(* IEC 61131-3 sources: crb-codesys/generation/scripts/repoeval/轴控/FB105_轴控制集/FB50_虚轴控制/FB104_全局变量2, 13 files *)

(* ---- G01_调模A轴.st ---- *)
VAR_GLOBAL
	FB_AxisControl_调模A轴: FB_轴控块;

//轴触发类
	b调模A轴正向点动: BOOL;
	b调模A轴反向点动: BOOL;
	b调模A轴正向寸动: BOOL;
	b调模A轴反向寸动: BOOL;
	b调模A轴停止触发: BOOL;
	b调模A轴复位触发: BOOL;
	b调模A轴绝对运动触发: BOOL;
	b调模A轴相对运动触发: BOOL;
	b调模A轴速度模式触发: BOOL;
	b调模A轴启用限位: BOOL;

//轴状态类
    b调模A轴通讯OK: BOOL;
	b调模A轴使能OK: BOOL;
	b调模A轴停止完成: BOOL;
	b调模A轴绝对运动完成: BOOL;
	b调模A轴相对运动完成: BOOL;
	b调模A轴速度模式Busy: BOOL;
	b调模A轴寸动模式Busy: BOOL;
	b调模A轴点动模式Busy: BOOL;
	b调模A轴绝对模式Busy: BOOL;
	b调模A轴相对模式Busy: BOOL;
	b调模A轴错误: BOOL;
	b调模A轴加速中: BOOL;
	b调模A轴减速中: BOOL;
    b调模A轴停止中: BOOL;

//数据给定类
	r调模A轴点动速度给定: LREAL;
	r调模A轴绝对运动速度给定: LREAL;
	r调模A轴相对运动速度给定: LREAL;
	r调模A轴速度模式速度给定: LREAL;
	r调模A轴寸动速度给定: LREAL;

	r调模A轴绝对运动位置给定: LREAL;
	r调模A轴相对运动位置给定: LREAL;
	r调模A轴寸动位置给定: LREAL;

//数据读取类
    r调模A轴当前位置: LREAL;
	r调模A轴当前速度: LREAL;
	r调模A轴当前扭矩: LREAL;

//其它类
    b调模A轴回零触发: BOOL;
    b调模A轴回零Busy: BOOL;
    b调模A轴回零完成: BOOL;
END_VAR

//HMI_PLC_BOOL映射
VAR_GLOBAL
	HMI_b调模A轴断使能 	 AT %MX300.0: BOOL;
	HMI_b调模A轴单独回原 AT %MX300.1: BOOL;
	HMI_b调模A轴正向点动 AT %MX300.2: BOOL;
    HMI_b调模A轴反向点动 AT %MX300.3: BOOL;

	HMI_b调模A轴去工作位 AT %MX300.4: BOOL;
END_VAR

//HMI_PLC_Data映射
VAR_GLOBAL PERSISTENT RETAIN
	HMI_r调模A轴当前位置 	AT %MD15600: REAL;
	HMI_r调模A轴当前速度 	AT %MD15601: REAL;
	HMI_r调模A轴自动速度 	AT %MD15602: REAL;
	HMI_r调模A轴手动速度 	AT %MD15603: REAL;

	HMI_r调模A轴导程 		AT %MD15604: REAL;
	HMI_r调模A轴齿轮比分子 	AT %MD15605: REAL;
	HMI_r调模A轴齿轮比分母 	AT %MD15606: REAL;

	HMI_r调模A轴回零快速 	AT %MD15607: REAL;
	HMI_r调模A轴回零慢速 	AT %MD15608: REAL;
	HMI_r调模A轴正限位 		AT %MD15609: REAL;
	HMI_r调模A轴负限位 		AT %MD15610: REAL;

	HMI_r调模A轴加速时间 	AT %MD15611: REAL;
	HMI_r调模A轴减速时间 	AT %MD15612: REAL;

	HMI_r调模A轴宽度位置 	AT %MD15613: REAL;

END_VAR

(* ---- G02_调模B轴.st ---- *)
VAR_GLOBAL
	FB_AxisControl_调模B轴: FB_轴控块;

//轴触发类
	b调模B轴正向点动: BOOL;
	b调模B轴反向点动: BOOL;
	b调模B轴正向寸动: BOOL;
	b调模B轴反向寸动: BOOL;
	b调模B轴停止触发: BOOL;
	b调模B轴复位触发: BOOL;
	b调模B轴绝对运动触发: BOOL;
	b调模B轴相对运动触发: BOOL;
	b调模B轴速度模式触发: BOOL;
	b调模B轴启用限位: BOOL;

//轴状态类
    b调模B轴通讯OK: BOOL;
	b调模B轴使能OK: BOOL;
	b调模B轴停止完成: BOOL;
	b调模B轴绝对运动完成: BOOL;
	b调模B轴相对运动完成: BOOL;
	b调模B轴速度模式Busy: BOOL;
	b调模B轴寸动模式Busy: BOOL;
	b调模B轴点动模式Busy: BOOL;
	b调模B轴绝对模式Busy: BOOL;
	b调模B轴相对模式Busy: BOOL;
	b调模B轴错误: BOOL;
	b调模B轴加速中: BOOL;
	b调模B轴减速中: BOOL;
    b调模B轴停止中: BOOL;

//数据给定类
	r调模B轴点动速度给定: LREAL;
	r调模B轴绝对运动速度给定: LREAL;
	r调模B轴相对运动速度给定: LREAL;
	r调模B轴速度模式速度给定: LREAL;
	r调模B轴寸动速度给定: LREAL;

	r调模B轴绝对运动位置给定: LREAL;
	r调模B轴相对运动位置给定: LREAL;
	r调模B轴寸动位置给定: LREAL;

//数据读取类
    r调模B轴当前位置: LREAL;
	r调模B轴当前速度: LREAL;
	r调模B轴当前扭矩: LREAL;

//其它类
    b调模B轴回零触发: BOOL;
    b调模B轴回零Busy: BOOL;
    b调模B轴回零完成: BOOL;
END_VAR

//HMI_PLC_BOOL映射
VAR_GLOBAL
	HMI_b调模B轴断使能 	 AT %MX305.0: BOOL;
	HMI_b调模B轴单独回原 AT %MX305.1: BOOL;
	HMI_b调模B轴正向点动 AT %MX305.2: BOOL;
    HMI_b调模B轴反向点动 AT %MX305.3: BOOL;

	HMI_b调模B轴去工作位 AT %MX305.4: BOOL;
END_VAR

//HMI_PLC_Data映射
VAR_GLOBAL
	HMI_r调模B轴当前位置 	AT %MD15650: REAL;
	HMI_r调模B轴当前速度 	AT %MD15651: REAL;
	HMI_r调模B轴自动速度 	AT %MD15652: REAL;
	HMI_r调模B轴手动速度 	AT %MD15653: REAL;

	HMI_r调模B轴导程 		AT %MD15654: REAL;
	HMI_r调模B轴齿轮比分子 	AT %MD15655: REAL;
	HMI_r调模B轴齿轮比分母 	AT %MD15656: REAL;

	HMI_r调模B轴回零快速 	AT %MD15657: REAL;
	HMI_r调模B轴回零慢速 	AT %MD15658: REAL;
	HMI_r调模B轴正限位 		AT %MD15659: REAL;
	HMI_r调模B轴负限位 		AT %MD15660: REAL;

	HMI_r调模B轴加速时间 	AT %MD15661: REAL;
	HMI_r调模B轴减速时间 	AT %MD15662: REAL;

	HMI_r调模B轴宽度位置 	AT %MD15663: REAL;
END_VAR

(* ---- G03_送面料轴.st ---- *)
VAR_GLOBAL
	FB_AxisControl_送面料轴: FB_轴控块;

//轴触发类
	b送面料轴正向点动: BOOL;
	b送面料轴反向点动: BOOL;
	b送面料轴正向寸动: BOOL;
	b送面料轴反向寸动: BOOL;
	b送面料轴停止触发: BOOL;
	b送面料轴复位触发: BOOL;
	b送面料轴绝对运动触发: BOOL;
	b送面料轴相对运动触发: BOOL;
	b送面料轴速度模式触发: BOOL;
	b送面料轴启用限位: BOOL;

//轴状态类
    b送面料轴通讯OK: BOOL;
	b送面料轴使能OK: BOOL;
	b送面料轴停止完成: BOOL;
	b送面料轴绝对运动完成: BOOL;
	b送面料轴相对运动完成: BOOL;
	b送面料轴速度模式Busy: BOOL;
	b送面料轴寸动模式Busy: BOOL;
	b送面料轴点动模式Busy: BOOL;
	b送面料轴绝对模式Busy: BOOL;
	b送面料轴相对模式Busy: BOOL;
	b送面料轴错误: BOOL;
	b送面料轴加速中: BOOL;
	b送面料轴减速中: BOOL;
    b送面料轴停止中: BOOL;

//数据给定类
	r送面料轴点动速度给定: LREAL;
	r送面料轴绝对运动速度给定: LREAL;
	r送面料轴相对运动速度给定: LREAL;
	r送面料轴速度模式速度给定: LREAL;
	r送面料轴寸动速度给定: LREAL;

	r送面料轴绝对运动位置给定: LREAL;
	r送面料轴相对运动位置给定: LREAL;
	r送面料轴寸动位置给定: LREAL;

//数据读取类
    r送面料轴当前位置: LREAL;
	r送面料轴当前速度: LREAL;
	r送面料轴当前扭矩: LREAL;

//其它类
    b送面料轴回零触发: BOOL;
    b送面料轴回零Busy: BOOL;
    b送面料轴回零完成: BOOL;
END_VAR

//HMI_PLC_BOOL映射
VAR_GLOBAL
	HMI_b送面料轴断使能 	 AT %MX310.0: BOOL;
	HMI_b送面料轴单独回原 	 AT %MX310.1: BOOL;
	HMI_b送面料轴正向点动 	 AT %MX310.2: BOOL;
    HMI_b送面料轴反向点动 	 AT %MX310.3: BOOL;

	HMI_b送面料轴设为原点 	 AT %MX310.4: BOOL;

	HMI_b送面料轴去停料位 	 	 AT %MX310.5: BOOL;
	HMI_b送面料轴去停料位保存 	 AT %MX310.6: BOOL;
END_VAR

//HMI_PLC_Data映射
VAR_GLOBAL
	HMI_r送面料轴当前位置 : REAL;
	HMI_r送面料轴当前速度 	AT %MD15700: REAL;
	HMI_r送面料轴自动速度 	AT %MD15701: REAL;
	HMI_r送面料轴手动速度 	AT %MD15702: REAL;

	HMI_r送面料轴导程 		AT %MD15703: REAL;
	HMI_r送面料轴齿轮比分子 AT %MD15704: REAL;
	HMI_r送面料轴齿轮比分母 AT %MD15705: REAL;

	HMI_r送面料轴回零快速 	AT %MD15706: REAL;
	HMI_r送面料轴回零慢速 	AT %MD15707: REAL;
	HMI_r送面料轴正限位 	AT %MD15708: REAL;
	HMI_r送面料轴负限位 	AT %MD15709: REAL;

	HMI_r送面料轴加速时间 	AT %MD15710: REAL;
	HMI_r送面料轴减速时间 	AT %MD15711: REAL;

	HMI_r送面料轴定位走距离长度 AT %MD15712: REAL;
	HMI_r送面料轴停料位 		AT %MD15713: REAL;

END_VAR

(* ---- G04_取面料轴.st ---- *)
VAR_GLOBAL
	FB_AxisControl_取面料轴: FB_轴控块;

//轴触发类
	b取面料轴正向点动: BOOL;
	b取面料轴反向点动: BOOL;
	b取面料轴正向寸动: BOOL;
	b取面料轴反向寸动: BOOL;
	b取面料轴停止触发: BOOL;
	b取面料轴复位触发: BOOL;
	b取面料轴绝对运动触发: BOOL;
	b取面料轴相对运动触发: BOOL;
	b取面料轴速度模式触发: BOOL;
	b取面料轴启用限位: BOOL;

//轴状态类
    b取面料轴通讯OK: BOOL;
	b取面料轴使能OK: BOOL;
	b取面料轴停止完成: BOOL;
	b取面料轴绝对运动完成: BOOL;
	b取面料轴相对运动完成: BOOL;
	b取面料轴速度模式Busy: BOOL;
	b取面料轴寸动模式Busy: BOOL;
	b取面料轴点动模式Busy: BOOL;
	b取面料轴绝对模式Busy: BOOL;
	b取面料轴相对模式Busy: BOOL;
	b取面料轴错误: BOOL;
	b取面料轴加速中: BOOL;
	b取面料轴减速中: BOOL;
    b取面料轴停止中: BOOL;

//数据给定类
	r取面料轴点动速度给定: LREAL;
	r取面料轴绝对运动速度给定: LREAL;
	r取面料轴相对运动速度给定: LREAL;
	r取面料轴速度模式速度给定: LREAL;
	r取面料轴寸动速度给定: LREAL;

	r取面料轴绝对运动位置给定: LREAL;
	r取面料轴相对运动位置给定: LREAL;
	r取面料轴寸动位置给定: LREAL;

//数据读取类
    r取面料轴当前位置: LREAL;
	r取面料轴当前速度: LREAL;
	r取面料轴当前扭矩: LREAL;

//其它类
    b取面料轴回零触发: BOOL;
    b取面料轴回零Busy: BOOL;
    b取面料轴回零完成: BOOL;
END_VAR

//HMI_PLC_BOOL映射
VAR_GLOBAL
	HMI_b取面料轴断使能 	 AT %MX315.0: BOOL;
	HMI_b取面料轴单独回原 	 AT %MX315.1: BOOL;
	HMI_b取面料轴正向点动 	 AT %MX315.2: BOOL;
    HMI_b取面料轴反向点动 	 AT %MX315.3: BOOL;

	HMI_b取面料轴设为原点 	 AT %MX315.4: BOOL;
	HMI_b取面料轴去取料位 	 AT %MX315.5: BOOL;
	HMI_b取面料轴去等待位 	 AT %MX315.6: BOOL;
	HMI_b取面料轴去送料位 	 AT %MX315.7: BOOL;
END_VAR

//HMI_PLC_Data映射
VAR_GLOBAL
	HMI_r取面料轴当前位置 	AT %MD15750: REAL;
	HMI_r取面料轴当前速度 	AT %MD15751: REAL;
	HMI_r取面料轴自动速度 	AT %MD15752: REAL;
	HMI_r取面料轴手动速度 	AT %MD15753: REAL;

	HMI_r取面料轴导程 		AT %MD15754: REAL;
	HMI_r取面料轴齿轮比分子 AT %MD15755: REAL;
	HMI_r取面料轴齿轮比分母 AT %MD15756: REAL;

	HMI_r取面料轴回零快速 	AT %MD15757: REAL;
	HMI_r取面料轴回零慢速 	AT %MD15758: REAL;
	HMI_r取面料轴正限位 	AT %MD15759: REAL;
	HMI_r取面料轴负限位 	AT %MD15760: REAL;

	HMI_r取面料轴加速时间 	AT %MD15761: REAL;
	HMI_r取面料轴减速时间 	AT %MD15762: REAL;

	HMI_r取面料轴取料位 	AT %MD15763: REAL;
	HMI_r取面料轴等待位 	AT %MD15764: REAL;
	HMI_r取面料轴送料位 	AT %MD15765: REAL;

END_VAR

(* ---- G05_横移A轴.st ---- *)
VAR_GLOBAL
	FB_AxisControl_横移A轴: FB_轴控块;

//轴触发类
	b横移A轴正向点动: BOOL;
	b横移A轴反向点动: BOOL;
	b横移A轴正向寸动: BOOL;
	b横移A轴反向寸动: BOOL;
	b横移A轴停止触发: BOOL;
	b横移A轴复位触发: BOOL;
	b横移A轴绝对运动触发: BOOL;
	b横移A轴相对运动触发: BOOL;
	b横移A轴速度模式触发: BOOL;
	b横移A轴启用限位: BOOL;

//轴状态类
    b横移A轴通讯OK: BOOL;
	b横移A轴使能OK: BOOL;
	b横移A轴停止完成: BOOL;
	b横移A轴绝对运动完成: BOOL;
	b横移A轴相对运动完成: BOOL;
	b横移A轴速度模式Busy: BOOL;
	b横移A轴寸动模式Busy: BOOL;
	b横移A轴点动模式Busy: BOOL;
	b横移A轴绝对模式Busy: BOOL;
	b横移A轴相对模式Busy: BOOL;
	b横移A轴错误: BOOL;
	b横移A轴加速中: BOOL;
	b横移A轴减速中: BOOL;
    b横移A轴停止中: BOOL;

//数据给定类
	r横移A轴点动速度给定: LREAL;
	r横移A轴绝对运动速度给定: LREAL;
	r横移A轴相对运动速度给定: LREAL;
	r横移A轴速度模式速度给定: LREAL;
	r横移A轴寸动速度给定: LREAL;

	r横移A轴绝对运动位置给定: LREAL;
	r横移A轴相对运动位置给定: LREAL;
	r横移A轴寸动位置给定: LREAL;

//数据读取类
    r横移A轴当前位置: LREAL;
	r横移A轴当前速度: LREAL;
	r横移A轴当前扭矩: LREAL;

//其它类
    b横移A轴回零触发: BOOL;
    b横移A轴回零Busy: BOOL;
    b横移A轴回零完成: BOOL;
END_VAR

//HMI_PLC_BOOL映射
VAR_GLOBAL
	HMI_b横移A轴断使能 	 AT %MX320.0: BOOL;
	HMI_b横移A轴单独回原 AT %MX320.1: BOOL;
	HMI_b横移A轴正向点动 AT %MX320.2: BOOL;
    HMI_b横移A轴反向点动 AT %MX320.3: BOOL;

	HMI_b横移A轴设为原点 AT %MX320.4: BOOL;
	HMI_b横移A轴去接底板位 AT %MX320.5: BOOL;
	HMI_b横移A轴去成型位 AT %MX320.6: BOOL;
END_VAR

//HMI_PLC_Data映射
VAR_GLOBAL
	HMI_r横移A轴当前位置 	AT %MD15800: REAL;
	HMI_r横移A轴当前速度 	AT %MD15801: REAL;
	HMI_r横移A轴自动速度 	AT %MD15802: REAL;
	HMI_r横移A轴手动速度 	AT %MD15803: REAL;

	HMI_r横移A轴导程 		AT %MD15804: REAL;
	HMI_r横移A轴齿轮比分子 	AT %MD15805: REAL;
	HMI_r横移A轴齿轮比分母 	AT %MD15806: REAL;

	HMI_r横移A轴回零快速 	AT %MD15807: REAL;
	HMI_r横移A轴回零慢速 	AT %MD15808: REAL;
	HMI_r横移A轴正限位 		AT %MD15809: REAL;
	HMI_r横移A轴负限位 		AT %MD15810: REAL;

	HMI_r横移A轴加速时间 	AT %MD15811: REAL;
	HMI_r横移A轴减速时间 	AT %MD15812: REAL;

	HMI_r横移A轴接底板位 	AT %MD15813: REAL;
	HMI_r横移A轴成型位 		AT %MD15814: REAL;

END_VAR

(* ---- G06_升降A轴.st ---- *)
VAR_GLOBAL
	FB_AxisControl_升降A轴: FB_轴控块;

//轴触发类
	b升降A轴正向点动: BOOL;
	b升降A轴反向点动: BOOL;
	b升降A轴正向寸动: BOOL;
	b升降A轴反向寸动: BOOL;
	b升降A轴停止触发: BOOL;
	b升降A轴复位触发: BOOL;
	b升降A轴绝对运动触发: BOOL;
	b升降A轴相对运动触发: BOOL;
	b升降A轴速度模式触发: BOOL;
	b升降A轴启用限位: BOOL;

//轴状态类
    b升降A轴通讯OK: BOOL;
	b升降A轴使能OK: BOOL;
	b升降A轴停止完成: BOOL;
	b升降A轴绝对运动完成: BOOL;
	b升降A轴相对运动完成: BOOL;
	b升降A轴速度模式Busy: BOOL;
	b升降A轴寸动模式Busy: BOOL;
	b升降A轴点动模式Busy: BOOL;
	b升降A轴绝对模式Busy: BOOL;
	b升降A轴相对模式Busy: BOOL;
	b升降A轴错误: BOOL;
	b升降A轴加速中: BOOL;
	b升降A轴减速中: BOOL;
    b升降A轴停止中: BOOL;

//数据给定类
	r升降A轴点动速度给定: LREAL;
	r升降A轴绝对运动速度给定: LREAL;
	r升降A轴相对运动速度给定: LREAL;
	r升降A轴速度模式速度给定: LREAL;
	r升降A轴寸动速度给定: LREAL;

	r升降A轴绝对运动位置给定: LREAL;
	r升降A轴相对运动位置给定: LREAL;
	r升降A轴寸动位置给定: LREAL;

//数据读取类
    r升降A轴当前位置: LREAL;
	r升降A轴当前速度: LREAL;
	r升降A轴当前扭矩: LREAL;

//其它类
    b升降A轴回零触发: BOOL;
    b升降A轴回零Busy: BOOL;
    b升降A轴回零完成: BOOL;
END_VAR

//HMI_PLC_BOOL映射
VAR_GLOBAL
	HMI_b升降A轴断使能 	 AT %MX325.0: BOOL;
	HMI_b升降A轴单独回原 AT %MX325.1: BOOL;
	HMI_b升降A轴正向点动 AT %MX325.2: BOOL;
    HMI_b升降A轴反向点动 AT %MX325.3: BOOL;

	HMI_b升降A轴设为原点 AT %MX325.4: BOOL;
	HMI_b升降A轴去接底板位 	 AT %MX325.5: BOOL;
	HMI_b升降A轴去接面位 	 AT %MX325.6: BOOL;
	HMI_b升降A轴去成型位 	 AT %MX325.7: BOOL;
	HMI_b升降A轴去出料位 	 AT %MX326.0: BOOL;
END_VAR

//HMI_PLC_Data映射
VAR_GLOBAL
	HMI_r升降A轴当前位置 	AT %MD15850: REAL;
	HMI_r升降A轴当前速度 	AT %MD15851: REAL;
	HMI_r升降A轴自动速度 	AT %MD15852: REAL;
	HMI_r升降A轴手动速度 	AT %MD15853: REAL;

	HMI_r升降A轴导程 		AT %MD15854: REAL;
	HMI_r升降A轴齿轮比分子 	AT %MD15855: REAL;
	HMI_r升降A轴齿轮比分母 	AT %MD15856: REAL;

	HMI_r升降A轴回零快速 	AT %MD15857: REAL;
	HMI_r升降A轴回零慢速 	AT %MD15858: REAL;
	HMI_r升降A轴正限位 		AT %MD15859: REAL;
	HMI_r升降A轴负限位 		AT %MD15860: REAL;

	HMI_r升降A轴加速时间 	AT %MD15861: REAL;
	HMI_r升降A轴减速时间 	AT %MD15862: REAL;

	HMI_r升降A轴接底板位 	AT %MD15863: REAL;
	HMI_r升降A轴接面位 		AT %MD15864: REAL;
	HMI_r升降A轴成型位 		AT %MD15865: REAL;
	HMI_r升降A轴出料位 		AT %MD15866: REAL;

END_VAR

(* ---- G07_横移B轴.st ---- *)
VAR_GLOBAL
	FB_AxisControl_横移B轴: FB_轴控块;

//轴触发类
	b横移B轴正向点动: BOOL;
	b横移B轴反向点动: BOOL;
	b横移B轴正向寸动: BOOL;
	b横移B轴反向寸动: BOOL;
	b横移B轴停止触发: BOOL;
	b横移B轴复位触发: BOOL;
	b横移B轴绝对运动触发: BOOL;
	b横移B轴相对运动触发: BOOL;
	b横移B轴速度模式触发: BOOL;
	b横移B轴启用限位: BOOL;

//轴状态类
    b横移B轴通讯OK: BOOL;
	b横移B轴使能OK: BOOL;
	b横移B轴停止完成: BOOL;
	b横移B轴绝对运动完成: BOOL;
	b横移B轴相对运动完成: BOOL;
	b横移B轴速度模式Busy: BOOL;
	b横移B轴寸动模式Busy: BOOL;
	b横移B轴点动模式Busy: BOOL;
	b横移B轴绝对模式Busy: BOOL;
	b横移B轴相对模式Busy: BOOL;
	b横移B轴错误: BOOL;
	b横移B轴加速中: BOOL;
	b横移B轴减速中: BOOL;
    b横移B轴停止中: BOOL;

//数据给定类
	r横移B轴点动速度给定: LREAL;
	r横移B轴绝对运动速度给定: LREAL;
	r横移B轴相对运动速度给定: LREAL;
	r横移B轴速度模式速度给定: LREAL;
	r横移B轴寸动速度给定: LREAL;

	r横移B轴绝对运动位置给定: LREAL;
	r横移B轴相对运动位置给定: LREAL;
	r横移B轴寸动位置给定: LREAL;

//数据读取类
    r横移B轴当前位置: LREAL;
	r横移B轴当前速度: LREAL;
	r横移B轴当前扭矩: LREAL;

//其它类
    b横移B轴回零触发: BOOL;
    b横移B轴回零Busy: BOOL;
    b横移B轴回零完成: BOOL;
END_VAR

//HMI_PLC_BOOL映射
VAR_GLOBAL
	HMI_b横移B轴断使能 	 	 AT %MX330.0: BOOL;
	HMI_b横移B轴单独回原 	 AT %MX330.1: BOOL;
	HMI_b横移B轴正向点动 	 AT %MX330.2: BOOL;
    HMI_b横移B轴反向点动 	 AT %MX330.3: BOOL;

	HMI_b横移B轴设为原点 	 AT %MX330.4: BOOL;
	HMI_b横移B轴去接底板位 	 AT %MX330.5: BOOL;
	HMI_b横移B轴去成型位 	 AT %MX330.6: BOOL;
END_VAR

//HMI_PLC_Data映射
VAR_GLOBAL
	HMI_r横移B轴当前位置 	AT %MD15900: REAL;
	HMI_r横移B轴当前速度 	AT %MD15901: REAL;
	HMI_r横移B轴自动速度 	AT %MD15902: REAL;
	HMI_r横移B轴手动速度 	AT %MD15903: REAL;

	HMI_r横移B轴导程 		AT %MD15904: REAL;
	HMI_r横移B轴齿轮比分子 	AT %MD15905: REAL;
	HMI_r横移B轴齿轮比分母 	AT %MD15906: REAL;

	HMI_r横移B轴回零快速 	AT %MD15907: REAL;
	HMI_r横移B轴回零慢速 	AT %MD15908: REAL;
	HMI_r横移B轴正限位 		AT %MD15909: REAL;
	HMI_r横移B轴负限位 		AT %MD15910: REAL;

	HMI_r横移B轴加速时间 	AT %MD15911: REAL;
	HMI_r横移B轴减速时间 	AT %MD15912: REAL;

	HMI_r横移B轴接底板位 	AT %MD15913: REAL;
	HMI_r横移B轴成型位 		AT %MD15914: REAL;

END_VAR

(* ---- G08_升降B轴.st ---- *)
VAR_GLOBAL
	FB_AxisControl_升降B轴: FB_轴控块;

//轴触发类
	b升降B轴正向点动: BOOL;
	b升降B轴反向点动: BOOL;
	b升降B轴正向寸动: BOOL;
	b升降B轴反向寸动: BOOL;
	b升降B轴停止触发: BOOL;
	b升降B轴复位触发: BOOL;
	b升降B轴绝对运动触发: BOOL;
	b升降B轴相对运动触发: BOOL;
	b升降B轴速度模式触发: BOOL;
	b升降B轴启用限位: BOOL;

//轴状态类
    b升降B轴通讯OK: BOOL;
	b升降B轴使能OK: BOOL;
	b升降B轴停止完成: BOOL;
	b升降B轴绝对运动完成: BOOL;
	b升降B轴相对运动完成: BOOL;
	b升降B轴速度模式Busy: BOOL;
	b升降B轴寸动模式Busy: BOOL;
	b升降B轴点动模式Busy: BOOL;
	b升降B轴绝对模式Busy: BOOL;
	b升降B轴相对模式Busy: BOOL;
	b升降B轴错误: BOOL;
	b升降B轴加速中: BOOL;
	b升降B轴减速中: BOOL;
    b升降B轴停止中: BOOL;

//数据给定类
	r升降B轴点动速度给定: LREAL;
	r升降B轴绝对运动速度给定: LREAL;
	r升降B轴相对运动速度给定: LREAL;
	r升降B轴速度模式速度给定: LREAL;
	r升降B轴寸动速度给定: LREAL;

	r升降B轴绝对运动位置给定: LREAL;
	r升降B轴相对运动位置给定: LREAL;
	r升降B轴寸动位置给定: LREAL;

//数据读取类
    r升降B轴当前位置: LREAL;
	r升降B轴当前速度: LREAL;
	r升降B轴当前扭矩: LREAL;

//其它类
    b升降B轴回零触发: BOOL;
    b升降B轴回零Busy: BOOL;
    b升降B轴回零完成: BOOL;
END_VAR

//HMI_PLC_BOOL映射
VAR_GLOBAL
	HMI_b升降B轴断使能 	 		AT %MX335.0: BOOL;
	HMI_b升降B轴单独回原 		AT %MX335.1: BOOL;
	HMI_b升降B轴正向点动 	 	AT %MX335.2: BOOL;
    HMI_b升降B轴反向点动 	 	AT %MX335.3: BOOL;

	HMI_b升降B轴设为原点 	 	AT %MX335.4: BOOL;
	HMI_b升降B轴去接底板位 	 	AT %MX335.5: BOOL;
	HMI_b升降B轴去接面位 	 	AT %MX335.6: BOOL;
	HMI_b升降B轴去成型位 	 	AT %MX335.7: BOOL;
	HMI_b升降B轴去出料位 	 	AT %MX336.0: BOOL;
END_VAR

//HMI_PLC_Data映射
VAR_GLOBAL
	HMI_r升降B轴当前位置 	AT %MD15950: REAL;
	HMI_r升降B轴当前速度 	AT %MD15951: REAL;
	HMI_r升降B轴自动速度 	AT %MD15952: REAL;
	HMI_r升降B轴手动速度 	AT %MD15953: REAL;

	HMI_r升降B轴导程 		AT %MD15954: REAL;
	HMI_r升降B轴齿轮比分子 	AT %MD15955: REAL;
	HMI_r升降B轴齿轮比分母 	AT %MD15956: REAL;

	HMI_r升降B轴回零快速 	AT %MD15957: REAL;
	HMI_r升降B轴回零慢速 	AT %MD15958: REAL;
	HMI_r升降B轴正限位 		AT %MD15959: REAL;
	HMI_r升降B轴负限位 		AT %MD15960: REAL;

	HMI_r升降B轴加速时间 	AT %MD15961: REAL;
	HMI_r升降B轴减速时间 	AT %MD15962: REAL;

	HMI_r升降B轴接底板位 	AT %MD15963: REAL;
	HMI_r升降B轴接面位 		AT %MD15964: REAL;
	HMI_r升降B轴成型位 		AT %MD15965: REAL;
	HMI_r升降B轴出料位 		AT %MD15966: REAL;
END_VAR

(* ---- G09_出盒轴.st ---- *)
VAR_GLOBAL
	FB_AxisControl_出盒轴: FB_轴控块;

//轴触发类
	b出盒轴正向点动: BOOL;
	b出盒轴反向点动: BOOL;
	b出盒轴正向寸动: BOOL;
	b出盒轴反向寸动: BOOL;
	b出盒轴停止触发: BOOL;
	b出盒轴复位触发: BOOL;
	b出盒轴绝对运动触发: BOOL;
	b出盒轴相对运动触发: BOOL;
	b出盒轴速度模式触发: BOOL;
	b出盒轴启用限位: BOOL;

//轴状态类
    b出盒轴通讯OK: BOOL;
	b出盒轴使能OK: BOOL;
	b出盒轴停止完成: BOOL;
	b出盒轴绝对运动完成: BOOL;
	b出盒轴相对运动完成: BOOL;
	b出盒轴速度模式Busy: BOOL;
	b出盒轴寸动模式Busy: BOOL;
	b出盒轴点动模式Busy: BOOL;
	b出盒轴绝对模式Busy: BOOL;
	b出盒轴相对模式Busy: BOOL;
	b出盒轴错误: BOOL;
	b出盒轴加速中: BOOL;
	b出盒轴减速中: BOOL;
    b出盒轴停止中: BOOL;

//数据给定类
	r出盒轴点动速度给定: LREAL;
	r出盒轴绝对运动速度给定: LREAL;
	r出盒轴相对运动速度给定: LREAL;
	r出盒轴速度模式速度给定: LREAL;
	r出盒轴寸动速度给定: LREAL;

	r出盒轴绝对运动位置给定: LREAL;
	r出盒轴相对运动位置给定: LREAL;
	r出盒轴寸动位置给定: LREAL;

//数据读取类
    r出盒轴当前位置: LREAL;
	r出盒轴当前速度: LREAL;
	r出盒轴当前扭矩: LREAL;

//其它类
    b出盒轴回零触发: BOOL;
    b出盒轴回零Busy: BOOL;
    b出盒轴回零完成: BOOL;
END_VAR

//HMI_PLC_BOOL映射
VAR_GLOBAL
	HMI_b出盒轴断使能	AT %MX340.0: BOOL;
	HMI_b出盒轴单独回原	AT %MX340.1: BOOL;
	HMI_b出盒轴正向点动	AT %MX340.2: BOOL;
    HMI_b出盒轴反向点动	AT %MX340.3: BOOL;

	HMI_b出盒轴设为原点	AT %MX340.4: BOOL;
	HMI_b出盒轴去待料位	AT %MX340.5: BOOL;
	HMI_b出盒轴去出盒位	AT %MX340.6: BOOL;
END_VAR

//HMI_PLC_Data映射
VAR_GLOBAL
	HMI_r出盒轴当前位置 	AT %MD16000: REAL;
	HMI_r出盒轴当前速度		AT %MD16001: REAL;
	HMI_r出盒轴自动速度 	AT %MD16002: REAL;
	HMI_r出盒轴手动速度 	AT %MD16003: REAL;

	HMI_r出盒轴导程 		AT %MD16004: REAL;
	HMI_r出盒轴齿轮比分子 	AT %MD16005: REAL;
	HMI_r出盒轴齿轮比分母 	AT %MD16006: REAL;

	HMI_r出盒轴回零快速 	AT %MD16007: REAL;
	HMI_r出盒轴回零慢速 	AT %MD16008: REAL;
	HMI_r出盒轴正限位 		AT %MD16009: REAL;
	HMI_r出盒轴负限位 		AT %MD16010: REAL;

	HMI_r出盒轴加速时间 	AT %MD16011: REAL;
	HMI_r出盒轴减速时间 	AT %MD16012: REAL;

	HMI_r出盒轴待料位 		AT %MD16013: REAL;
	HMI_r出盒轴出盒位 		AT %MD16014: REAL;

END_VAR

(* ---- G10_铲灰板轴.st ---- *)
VAR_GLOBAL
	FB_AxisControl_铲灰板轴: FB_轴控块;

//轴触发类
	b铲灰板轴正向点动: BOOL;
	b铲灰板轴反向点动: BOOL;
	b铲灰板轴正向寸动: BOOL;
	b铲灰板轴反向寸动: BOOL;
	b铲灰板轴停止触发: BOOL;
	b铲灰板轴复位触发: BOOL;
	b铲灰板轴绝对运动触发: BOOL;
	b铲灰板轴相对运动触发: BOOL;
	b铲灰板轴速度模式触发: BOOL;
	b铲灰板轴启用限位: BOOL;

//轴状态类
    b铲灰板轴通讯OK: BOOL;
	b铲灰板轴使能OK: BOOL;
	b铲灰板轴停止完成: BOOL;
	b铲灰板轴绝对运动完成: BOOL;
	b铲灰板轴相对运动完成: BOOL;
	b铲灰板轴速度模式Busy: BOOL;
	b铲灰板轴寸动模式Busy: BOOL;
	b铲灰板轴点动模式Busy: BOOL;
	b铲灰板轴绝对模式Busy: BOOL;
	b铲灰板轴相对模式Busy: BOOL;
	b铲灰板轴错误: BOOL;
	b铲灰板轴加速中: BOOL;
	b铲灰板轴减速中: BOOL;
    b铲灰板轴停止中: BOOL;

//数据给定类
	r铲灰板轴点动速度给定: LREAL;
	r铲灰板轴绝对运动速度给定: LREAL;
	r铲灰板轴相对运动速度给定: LREAL;
	r铲灰板轴速度模式速度给定: LREAL;
	r铲灰板轴寸动速度给定: LREAL;

	r铲灰板轴绝对运动位置给定: LREAL;
	r铲灰板轴相对运动位置给定: LREAL;
	r铲灰板轴寸动位置给定: LREAL;

//数据读取类
    r铲灰板轴当前位置: LREAL;
	r铲灰板轴当前速度: LREAL;
	r铲灰板轴当前扭矩: LREAL;

//其它类
    b铲灰板轴回零触发: BOOL;
    b铲灰板轴回零Busy: BOOL;
    b铲灰板轴回零完成: BOOL;
END_VAR

//HMI_PLC_BOOL映射
VAR_GLOBAL
	HMI_b铲灰板轴断使能		AT %MX345.0: BOOL;
	HMI_b铲灰板轴单独回原	AT %MX345.1: BOOL;
	HMI_b铲灰板轴正向点动	AT %MX345.2: BOOL;
    HMI_b铲灰板轴反向点动	AT %MX345.3: BOOL;

	HMI_b铲灰板轴设为原点	AT %MX345.4: BOOL;
	HMI_b铲灰板轴去铲出位	AT %MX345.5: BOOL;
END_VAR

//HMI_PLC_Data映射
VAR_GLOBAL
	HMI_r铲灰板轴当前位置 	AT %MD16050: REAL;
	HMI_r铲灰板轴当前速度 	AT %MD16051: REAL;
	HMI_r铲灰板轴自动速度 	AT %MD16052: REAL;
	HMI_r铲灰板轴手动速度 	AT %MD16053: REAL;

	HMI_r铲灰板轴导程 		AT %MD16054: REAL;
	HMI_r铲灰板轴齿轮比分子 AT %MD16055: REAL;
	HMI_r铲灰板轴齿轮比分母 AT %MD16056: REAL;

	HMI_r铲灰板轴回零快速 	AT %MD16057: REAL;
	HMI_r铲灰板轴回零慢速 	AT %MD16058: REAL;
	HMI_r铲灰板轴正限位 	AT %MD16059: REAL;
	HMI_r铲灰板轴负限位 	AT %MD16060: REAL;

	HMI_r铲灰板轴加速时间 	AT %MD16061: REAL;
	HMI_r铲灰板轴减速时间 	AT %MD16062: REAL;

	HMI_r铲灰板轴铲出位 	AT %MD16063: REAL;

END_VAR

(* ---- G11_包面纸轴.st ---- *)
VAR_GLOBAL
	FB_AxisControl_包面纸轴: FB_轴控块;

//轴触发类
	b包面纸轴正向点动: BOOL;
	b包面纸轴反向点动: BOOL;
	b包面纸轴正向寸动: BOOL;
	b包面纸轴反向寸动: BOOL;
	b包面纸轴停止触发: BOOL;
	b包面纸轴复位触发: BOOL;
	b包面纸轴绝对运动触发: BOOL;
	b包面纸轴相对运动触发: BOOL;
	b包面纸轴速度模式触发: BOOL;
	b包面纸轴启用限位: BOOL;

//轴状态类
    b包面纸轴通讯OK: BOOL;
	b包面纸轴使能OK: BOOL;
	b包面纸轴停止完成: BOOL;
	b包面纸轴绝对运动完成: BOOL;
	b包面纸轴相对运动完成: BOOL;
	b包面纸轴速度模式Busy: BOOL;
	b包面纸轴寸动模式Busy: BOOL;
	b包面纸轴点动模式Busy: BOOL;
	b包面纸轴绝对模式Busy: BOOL;
	b包面纸轴相对模式Busy: BOOL;
	b包面纸轴错误: BOOL;
	b包面纸轴加速中: BOOL;
	b包面纸轴减速中: BOOL;
    b包面纸轴停止中: BOOL;

//数据给定类
	r包面纸轴点动速度给定: LREAL;
	r包面纸轴绝对运动速度给定: LREAL;
	r包面纸轴相对运动速度给定: LREAL;
	r包面纸轴速度模式速度给定: LREAL;
	r包面纸轴寸动速度给定: LREAL;

	r包面纸轴绝对运动位置给定: LREAL;
	r包面纸轴相对运动位置给定: LREAL;
	r包面纸轴寸动位置给定: LREAL;

//数据读取类
    r包面纸轴当前位置: LREAL;
	r包面纸轴当前速度: LREAL;
	r包面纸轴当前扭矩: LREAL;

//其它类
    b包面纸轴回零触发: BOOL;
    b包面纸轴回零Busy: BOOL;
    b包面纸轴回零完成: BOOL;
END_VAR

//HMI_PLC_BOOL映射
VAR_GLOBAL
	HMI_b包面纸轴断使能		AT %MX350.0: BOOL;
	HMI_b包面纸轴单独回原	AT %MX350.1: BOOL;
	HMI_b包面纸轴正向点动	AT %MX350.2: BOOL;
    HMI_b包面纸轴反向点动	AT %MX350.3: BOOL;

	HMI_b包面纸轴设为原点	AT %MX350.4: BOOL;
	HMI_b包面纸轴去包面位	AT %MX350.5: BOOL;
END_VAR

//HMI_PLC_Data映射
VAR_GLOBAL
	HMI_r包面纸轴当前位置 	AT %MD16100: REAL;
	HMI_r包面纸轴当前速度 	AT %MD16101: REAL;
	HMI_r包面纸轴自动速度 	AT %MD16102: REAL;
	HMI_r包面纸轴手动速度 	AT %MD16103: REAL;

	HMI_r包面纸轴导程 		AT %MD16104: REAL;
	HMI_r包面纸轴齿轮比分子 AT %MD16105: REAL;
	HMI_r包面纸轴齿轮比分母 AT %MD16106: REAL;

	HMI_r包面纸轴回零快速 	AT %MD16107: REAL;
	HMI_r包面纸轴回零慢速 	AT %MD16108: REAL;
	HMI_r包面纸轴正限位 	AT %MD16109: REAL;
	HMI_r包面纸轴负限位 	AT %MD16110: REAL;

	HMI_r包面纸轴加速时间 	AT %MD16111: REAL;
	HMI_r包面纸轴减速时间 	AT %MD16112: REAL;

	HMI_r包面纸轴包面位 	AT %MD16113: REAL;
END_VAR

(* ---- G12_上包底轴.st ---- *)
VAR_GLOBAL
	FB_AxisControl_上包底轴: FB_轴控块;

//轴触发类
	b上包底轴正向点动: BOOL;
	b上包底轴反向点动: BOOL;
	b上包底轴正向寸动: BOOL;
	b上包底轴反向寸动: BOOL;
	b上包底轴停止触发: BOOL;
	b上包底轴复位触发: BOOL;
	b上包底轴绝对运动触发: BOOL;
	b上包底轴相对运动触发: BOOL;
	b上包底轴速度模式触发: BOOL;
	b上包底轴启用限位: BOOL;

//轴状态类
    b上包底轴通讯OK: BOOL;
	b上包底轴使能OK: BOOL;
	b上包底轴停止完成: BOOL;
	b上包底轴绝对运动完成: BOOL;
	b上包底轴相对运动完成: BOOL;
	b上包底轴速度模式Busy: BOOL;
	b上包底轴寸动模式Busy: BOOL;
	b上包底轴点动模式Busy: BOOL;
	b上包底轴绝对模式Busy: BOOL;
	b上包底轴相对模式Busy: BOOL;
	b上包底轴错误: BOOL;
	b上包底轴加速中: BOOL;
	b上包底轴减速中: BOOL;
    b上包底轴停止中: BOOL;

//数据给定类
	r上包底轴点动速度给定: LREAL;
	r上包底轴绝对运动速度给定: LREAL;
	r上包底轴相对运动速度给定: LREAL;
	r上包底轴速度模式速度给定: LREAL;
	r上包底轴寸动速度给定: LREAL;

	r上包底轴绝对运动位置给定: LREAL;
	r上包底轴相对运动位置给定: LREAL;
	r上包底轴寸动位置给定: LREAL;

//数据读取类
    r上包底轴当前位置: LREAL;
	r上包底轴当前速度: LREAL;
	r上包底轴当前扭矩: LREAL;

//其它类
    b上包底轴回零触发: BOOL;
    b上包底轴回零Busy: BOOL;
    b上包底轴回零完成: BOOL;
END_VAR

//HMI_PLC_BOOL映射
VAR_GLOBAL
	HMI_b上包底轴断使能		AT %MX355.0: BOOL;
	HMI_b上包底轴单独回原	AT %MX355.1: BOOL;
	HMI_b上包底轴正向点动	AT %MX355.2: BOOL;
    HMI_b上包底轴反向点动	AT %MX355.3: BOOL;

	HMI_b上包底轴设为原点	AT %MX355.4: BOOL;
	HMI_b上包底轴去接底板位	AT %MX355.5: BOOL;
	HMI_b上包底轴去送底板位	AT %MX355.6: BOOL;
	HMI_b上包底轴去送等待位	AT %MX355.7: BOOL;

	HMI_b上包底轴去送底板A位 AT %MX356.0: BOOL;
	HMI_b上包底轴去送底板B位 AT %MX356.1: BOOL;
END_VAR

//HMI_PLC_Data映射
VAR_GLOBAL
	HMI_r上包底轴当前位置 	AT %MD16150: REAL;
	HMI_r上包底轴当前速度 	AT %MD16151: REAL;
	HMI_r上包底轴自动速度 	AT %MD16152: REAL;
	HMI_r上包底轴手动速度 	AT %MD16153: REAL;

	HMI_r上包底轴导程 		AT %MD16154: REAL;
	HMI_r上包底轴齿轮比分子 AT %MD16155: REAL;
	HMI_r上包底轴齿轮比分母 AT %MD16156: REAL;

	HMI_r上包底轴回零快速 	AT %MD16157: REAL;
	HMI_r上包底轴回零慢速 	AT %MD16158: REAL;
	HMI_r上包底轴正限位 	AT %MD16159: REAL;
	HMI_r上包底轴负限位 	AT %MD16160: REAL;

	HMI_r上包底轴加速时间	AT %MD16161: REAL;
	HMI_r上包底轴减速时间	AT %MD16162: REAL;

	HMI_r上包底轴接底板位	AT %MD16163: REAL;
	HMI_r上包底轴送底板位	AT %MD16164: REAL;
	HMI_r上包底轴送等待位	AT %MD16165: REAL;

	HMI_r上包底轴送底板A位	AT %MD16166: REAL;
	HMI_r上包底轴送底板B位	AT %MD16167: REAL;

END_VAR

(* ---- G13_折边轴.st ---- *)
VAR_GLOBAL
	FB_AxisControl_折边轴: FB_轴控块;

//轴触发类
	b折边轴正向点动: BOOL;
	b折边轴反向点动: BOOL;
	b折边轴正向寸动: BOOL;
	b折边轴反向寸动: BOOL;
	b折边轴停止触发: BOOL;
	b折边轴复位触发: BOOL;
	b折边轴绝对运动触发: BOOL;
	b折边轴相对运动触发: BOOL;
	b折边轴速度模式触发: BOOL;
	b折边轴启用限位: BOOL;

//轴状态类
    b折边轴通讯OK: BOOL;
	b折边轴使能OK: BOOL;
	b折边轴停止完成: BOOL;
	b折边轴绝对运动完成: BOOL;
	b折边轴相对运动完成: BOOL;
	b折边轴速度模式Busy: BOOL;
	b折边轴寸动模式Busy: BOOL;
	b折边轴点动模式Busy: BOOL;
	b折边轴绝对模式Busy: BOOL;
	b折边轴相对模式Busy: BOOL;
	b折边轴错误: BOOL;
	b折边轴加速中: BOOL;
	b折边轴减速中: BOOL;
    b折边轴停止中: BOOL;

//数据给定类
	r折边轴点动速度给定: LREAL;
	r折边轴绝对运动速度给定: LREAL;
	r折边轴相对运动速度给定: LREAL;
	r折边轴速度模式速度给定: LREAL;
	r折边轴寸动速度给定: LREAL;

	r折边轴绝对运动位置给定: LREAL;
	r折边轴相对运动位置给定: LREAL;
	r折边轴寸动位置给定: LREAL;

//数据读取类
    r折边轴当前位置: LREAL;
	r折边轴当前速度: LREAL;
	r折边轴当前扭矩: LREAL;

//其它类
    b折边轴回零触发: BOOL;
    b折边轴回零Busy: BOOL;
    b折边轴回零完成: BOOL;
END_VAR

//HMI_PLC_BOOL映射
VAR_GLOBAL
	HMI_b折边轴断使能	AT %MX360.0: BOOL;
	HMI_b折边轴单独回原	AT %MX360.1: BOOL;
	HMI_b折边轴正向点动	AT %MX360.2: BOOL;
    HMI_b折边轴反向点动	AT %MX360.3: BOOL;

	HMI_b折边轴设为原点	AT %MX360.4: BOOL;
	HMI_b折边轴去停料位	AT %MX360.5: BOOL;
END_VAR

//HMI_PLC_Data映射
VAR_GLOBAL
	HMI_r折边轴当前位置 	AT %MD16200: REAL;
	HMI_r折边轴当前速度 	AT %MD16201: REAL;
	HMI_r折边轴自动速度 	AT %MD16202: REAL;
	HMI_r折边轴手动速度 	AT %MD16203: REAL;

	HMI_r折边轴导程 		AT %MD16204: REAL;
	HMI_r折边轴齿轮比分子 	AT %MD16205: REAL;
	HMI_r折边轴齿轮比分母 	AT %MD16206: REAL;

	HMI_r折边轴回零快速 	AT %MD16207: REAL;
	HMI_r折边轴回零慢速 	AT %MD16208: REAL;
	HMI_r折边轴正限位 		AT %MD16209: REAL;
	HMI_r折边轴负限位 		AT %MD16210: REAL;

	HMI_r折边轴加速时间 	AT %MD16211: REAL;
	HMI_r折边轴减速时间 	AT %MD16212: REAL;

	HMI_r折边轴停料位 		AT %MD16213: REAL;
END_VAR
